{attribute 'hide_all_locals'}
FUNCTION_BLOCK FB_ECS_HTTP_ZaptecAccount
VAR_INPUT
	bStart					: BOOL;													//Start/Stop this Functions
	byMode					: BYTE;													//Work mode : 0 = Send current to each Charger; 1 = Send current to a Installation of chargers
	sUsername				: STRING(100);											//Username from the Zaptec Account
	sPassword				: STRING(100);											//Password from the Zaptec Account
	arrCharger				: ARRAY[1..100] OF ST_Zaptec_Input_Charger;				//Structure with Data for each Charging Station
	arrInstallation			: ARRAY[1..100] OF ST_Zaptec_Input_Installation;		//Structure with Data for each Installation of Charging Stations
END_VAR
VAR_OUTPUT
	bValidResult			: BOOL;													//Valid Result received from Server
	bBusy             		: BOOL;													//Busy Flag
    bError              	: BOOL;													//Error Flag
	hrErrorCode       		: HRESULT;												//Error Result from Http Client
	arrStateCharger			: ARRAY[1..100] OF ST_Zaptec_ECS_State;					//Output Structure with the State from each Charging Station
END_VAR
VAR
	fbHttpClient        	: FB_IotHttpClient :=(sHostName:='api.zaptec.com',		//Http Client Function
                       		  bKeepAlive:=FALSE, tConnectionTimeout:=T#10S);
	fbHttpPostToken         : FB_HTTP_Post_Zaptec_ReqToken;							//Http Post to receive the Bearer Token
 	fbHttpGetChrgState		: FB_HTTP_Get_Zaptec_ECS_State;							//Http Get to receive the State from each Charging station
	fbHttpPostCurrent		: FB_HTTP_Post_Zaptec_Current;							//Http Post to control each Chrging station or a installation of charging stations with the current setpoint
	fbTaskIndex				: GETCURTASKINDEX;										//Function to find the Task Index
	timDelay				: TON;													//Timer for Delay between the Requests
	timTimout				: TON;													//Timer for Timeout in the State machine
	timToken				: TON;													//Timer to make a Request for a new Token
	FPStart					: R_TRIG;												//Internal positive Edge
	FPErrorToken			: R_TRIG;												//Internal positive Edge
	FPErrorGetState			: R_TRIG;												//Internal positive Edge
	FPErrorPostCurrent		: R_TRIG;												//Internal positive Edge
	FPErrorClient			: R_TRIG;												//Internal positive Edge
	FPTimToken				: R_TRIG;												//Internal positive Edge
	FNStart					: F_TRIG;												//Internal negative Edge
	byNumberOfChargers		: BYTE;													//Number of charging station with insert ID in the Input Array
	byNumberOfInstallation	: BYTE;													//Number of Installations with insert ID in the Input Array
	byECSInProgress			: BYTE;													//Charging station in Progress to read out the State or write the current
	byInstInProgress		: BYTE;													//Installation of charging stations in Progress to write the current
	byLPInfo				: BYTE;													//Loop Variable to define some parts in the Code
	iState					: INT;													//Variabel for state machine
	iState_CP				: INT;													//Variabel for state machine to compare it for timeout
	udiCycleTime			: UDINT;												//Cycletime in ms
END_VAR

//Creator : Kai Ebensperger
//Company : Lynus AG
//Date : 04.11.2021
//Version : 1.0.0.0

//With this Function its possible to receive information from each charging station in a Zaptec Account in there cloudplattform
//Its also possible to control the charging station with this function by a curretn setpoint.
//We can control each Cahrging station with the current or each installation with more charging stations with a sum of current
//When the Installation mode is active, then the system of the charging station distribute the sum of current among themselves
//Attention : This Function need allways the Charging IDs. Even if the current is sent to the installation. Becasue the State Get Request for each charging station its possible only with the Charging IDs
//This Function can handle maximal 100 charging stations and 100 Installations

(*------------------------------------------------------------------------------------Limits------------------------------------------------------------------------------------------------------*)

byMode := LIMIT(0,byMode,1);

(*------------------------------------------------------------------------------------Configure HTTP Client------------------------------------------------------------------------------------------------------*)

IF NOT fbHttpClient.bConfigured THEN
    fbHttpClient.nHostPort:= 443;
	fbHttpClient.stTLS.bNoServerCertCheck := TRUE;
END_IF

(*------------------------------------------------------------------------------------Logic------------------------------------------------------------------------------------------------------*)

//Calculate the number of chargers and installations from the input array
byNumberOfChargers := 0;
	byNumberOfInstallation := 0;

FOR byLPInfo := 1 TO 100 BY 1 DO
	IF arrCharger[byLPInfo].sChargerID <> '' THEN byNumberOfChargers := byNumberOfChargers + 1; END_IF 
		IF arrInstallation[byLPInfo].sInstallationID <> '' THEN byNumberOfInstallation := byNumberOfInstallation + 1; END_IF  
END_FOR 	

//Delay between the Requests
fbTaskIndex(index=> );
	udiCycleTime := TwinCAT_SystemInfoVarList._TaskInfo[fbTaskIndex.index].CycleTime / 10000;
		timDelay(IN:= , PT:= T#1MS * udiCycleTime, Q=> , ET=> );

//Timout
IF iState_CP = iState AND iState <> 0 THEN timTimout.IN := TRUE; ELSE timTimout.IN := FALSE; END_IF
	timTimout(IN:= , PT:= T#20S, Q=> , ET=> );

//Timer for the Token
//After received the validation from the Token start this timer.
//After the Delay stop the State machine and make a request for a new Token
IF fbHttpPostToken.udiValidityToken <> 0 THEN
	timToken.PT := (T#1S * (fbHttpPostToken.udiValidityToken - 600));	//Less 10 Minutes
ELSE
	timToken.PT := T#600S;
END_IF
	timToken(IN:= , PT:= , Q=> , ET=> );	

FPTimToken(CLK:= timToken.Q, Q=> );
	
//Start	
FPStart(CLK:= bStart, Q=> );
	IF FPStart.Q AND NOT fbHttpPostToken.bBusy AND NOT fbHttpGetChrgState.bBusy AND NOT fbHttpPostCurrent.bBusy AND fbHttpClient.bConfigured THEN istate := 1; END_IF
		IF NOT bStart THEN istate := 0; END_IF	

CASE iState OF

	0://Init Step	
		fbHttpPostToken.bPostToken := FALSE;
			fbHttpGetChrgState.bSend := FALSE;
				fbHttpPostCurrent.bSend := FALSE;	
					byECSInProgress := 0;
						byInstInProgress := 0;
							timToken.IN := FALSE;
								bValidResult := FALSE;
									timdelay.IN := FALSE;
		
		FOR byLPInfo := 1 TO 100 BY 1 DO					
			arrStateCharger[byLPInfo].bIsEnabled := FALSE;	
				arrStateCharger[byLPInfo].bIsOnline := FALSE;
					arrStateCharger[byLPInfo].diOperationMode := 0;	
						arrStateCharger[byLPInfo].diWarnings := 0;
							arrStateCharger[byLPInfo].rAllocatedCurrent := 0;
								arrStateCharger[byLPInfo].rMaxCurrect := 0;
									arrStateCharger[byLPInfo].rMinCurrect := 0;
										arrStateCharger[byLPInfo].rCurrentL1 := 0;	
											arrStateCharger[byLPInfo].rCurrentL2 := 0;	
												arrStateCharger[byLPInfo].rCurrentL3 := 0;	
													arrStateCharger[byLPInfo].rPower := 0;
														arrStateCharger[byLPInfo].rEnergySession := 0;		
															arrStateCharger[byLPInfo].sChargerID := '';	
		END_FOR		
				
	1://Request for Bearer Token
		iState_CP := iState;
	
		fbHttpPostToken.bPostToken := TRUE;
			timToken.IN := FALSE;
		
		IF NOT fbHttpPostToken.bBusy THEN timdelay.IN := TRUE; END_IF 
	
		IF NOT fbHttpPostToken.bBusy AND fbHttpPostToken.bValidResult AND NOT fbHttpPostToken.bError AND timdelay.Q THEN
			istate := 2; 
				timdelay.IN := FALSE;
					byECSInProgress := 1;
						byInstInProgress := 1;
							fbHttpPostToken.bPostToken := FALSE;
								timToken.IN := TRUE;
		END_IF
		
		//Valid Result
		bValidResult := fbHttpPostToken.bValidResult;
		
		//Error, Timout or Request for a new Token
		IF FPErrorToken.Q OR timTimout.Q OR FPTimToken.Q OR FPErrorClient.Q THEN istate := 300; END_IF

	2://Request for State of Each Charging Station
		iState_CP := iState;
		
		fbHttpGetChrgState.bSend := TRUE;
			fbHttpGetChrgState.sChargerID := arrCharger[byECSInProgress].sChargerID;
		
		IF NOT fbHttpGetChrgState.bBusy THEN timdelay.IN := TRUE; END_IF 
		
		IF NOT fbHttpGetChrgState.bBusy AND fbHttpGetChrgState.bValidResult AND NOT fbHttpGetChrgState.bError AND timdelay.Q THEN
			IF byMode = 0 THEN istate := 3; END_IF
				IF byMode = 1 THEN istate := 4; END_IF
					timdelay.IN := FALSE;
						arrStateCharger[byECSInProgress] := fbHttpGetChrgState.stChargerStates;
							fbHttpGetChrgState.bSend := FALSE;	
		END_IF
		
		//Valid Result
		bValidResult := fbHttpGetChrgState.bValidResult;
		
		//Error, Timout or Request for a new Token
		IF FPErrorGetState.Q OR timTimout.Q OR FPTimToken.Q OR FPErrorClient.Q THEN istate := 300; END_IF
		
	3://Write current to charging station
		iState_CP := iState;
		
		fbHttpPostCurrent.bSend := TRUE;
			fbHttpPostCurrent.sID := arrCharger[byECSInProgress].sChargerID;
				fbHttpPostCurrent.rMaxCurrentCharger := arrCharger[byECSInProgress].rMaxCurrentCharger;
 					fbHttpPostCurrent.rMinCurrentCharger := arrCharger[byECSInProgress].rMinCurrentCharger;
		
		IF NOT fbHttpPostCurrent.bBusy THEN timdelay.IN := TRUE; END_IF 
		
		IF NOT fbHttpPostCurrent.bBusy AND fbHttpPostCurrent.bValidResult AND NOT fbHttpPostCurrent.bError AND timdelay.Q THEN
			iState := 5;
				timdelay.IN := FALSE;
					fbHttpPostCurrent.bSend := FALSE;	
		END_IF
		
		//Valid Result
		bValidResult := fbHttpPostCurrent.bValidResult;
		
		//Error, Timout or Request for a new Token
		IF FPErrorPostCurrent.Q OR timTimout.Q OR FPTimToken.Q OR FPErrorClient.Q THEN istate := 300; END_IF
		
	4://Write current to installation of charging stations	
		iState_CP := iState;	
	
		fbHttpPostCurrent.bSend := TRUE;
			fbHttpPostCurrent.sID := arrInstallation[byInstInProgress].sInstallationID;
				fbHttpPostCurrent.rAvailableCurrentInstallation := arrInstallation[byInstInProgress].rAvailableCurrentInstallation;
		
		IF NOT fbHttpPostCurrent.bBusy THEN timdelay.IN := TRUE; END_IF 
		
		IF NOT fbHttpPostCurrent.bBusy AND fbHttpPostCurrent.bValidResult AND NOT fbHttpPostCurrent.bError AND timdelay.Q THEN
			iState := 5;
				timdelay.IN := FALSE;
					fbHttpPostCurrent.bSend := FALSE;	
		END_IF
		
		//Valid Result
		bValidResult := fbHttpPostCurrent.bValidResult;
		
		//Error, Timout or Request for a new Token
		IF FPErrorPostCurrent.Q OR timTimout.Q OR FPTimToken.Q OR FPErrorClient.Q THEN istate := 300; END_IF
		
	5://Next charging station and next installation	
		iState_CP := iState;
		
		byECSInProgress := byECSInProgress + 1;
		byInstInProgress := byInstInProgress + 1;
		
		//Back to read out next state from charging station
		iState := 2;
		
		IF byECSInProgress > byNumberOfChargers THEN byECSInProgress := 1; END_IF
			IF byInstInProgress > byNumberOfInstallation THEN byInstInProgress := 1; END_IF  	
		
		//Reset Error
		bError := FALSE;
			
	300://Error or restart after receive a new Token
		iState_CP := iState;
		
		timdelay.IN := FALSE;
			fbHttpPostToken.bPostToken := FALSE;
				fbHttpGetChrgState.bSend := FALSE;
					fbHttpPostCurrent.bSend := FALSE;	
						byECSInProgress := 0;
							byInstInProgress := 0;
								bError := TRUE;
								//Restart
								IF NOT fbHttpPostToken.bBusy AND NOT fbHttpGetChrgState.bBusy AND NOT fbHttpPostCurrent.bBusy THEN 
									istate := 1;
								END_IF	
		
		
END_CASE		
		
(*------------------------------------------------------------------------------------HTTP Functions------------------------------------------------------------------------------------------------------*)

fbHttpPostToken(
	sUsername:= sUsername, 
	sPassword:= sPassword, 
	bPostToken:= , 
	tTimeOut:= T#20S,
	fbClient:= fbHttpClient, 
	bValidResult=> , 
	bBusy=> , 
	bError=> , 
	udiValidityToken=> , 
	sToken=> , 
	sTokenType=> );

FPErrorToken(CLK:= fbHttpPostToken.bError, Q=> );
	
fbHttpGetChrgState(
	bSend:= , 
	sToken:= fbHttpPostToken.sToken, 
	sTokenType:= fbHttpPostToken.sTokenType, 
	sChargerID:= , 
	tTimeOut:= T#20S,
	fbClient:= fbHttpClient, 
	bValidResult=> , 
	bBusy=> , 
	bError=> , 
	stChargerStates=> );

FPErrorGetState(CLK:= fbHttpGetChrgState.bError, Q=> );
	
fbHttpPostCurrent(
	bSend:= , 
	byMode:= byMode, 
	rMaxCurrentCharger:= , 
	rMinCurrentCharger:= , 
	rAvailableCurrentInstallation:= , 
	sToken:= fbHttpPostToken.sToken, 
	sTokenType:= fbHttpPostToken.sTokenType, 
	sID:= , 
	tTimeOut:= T#20S,
	fbClient:= fbHttpClient, 
	bValidResult=> , 
	bBusy=> , 
	bError=> );

FPErrorPostCurrent(CLK:= fbHttpPostCurrent.bError, Q=> );	

//Http Client
FNStart(CLK:= bStart, Q=> );
	IF FNStart.Q THEN fbHttpClient.Disconnect(); END_IF

fbHttpClient.Execute();

FPErrorClient(CLK:= fbHttpClient.bError, Q=> );

//Busy
IF fbHttpPostToken.bBusy OR fbHttpGetChrgState.bBusy OR fbHttpPostCurrent.bBusy THEN bBusy := TRUE; ELSE bBusy := FALSE; END_IF  

//Error
hrErrorCode := fbHttpClient.hrErrorCode;

END_FUNCTION_BLOCK

(* stored: Version 1.1.0.1, ProductVersion 3.1.4024.9
   POU FB_ECS_HTTP_ZaptecAccount: Id {5a052ac1-11ad-4d1b-9329-daffc7fe882a}, SpecialFunc None *)
